Staubli VAL3: InitBelt.pgx

program InitBelt()
begin
  //砂带信息初始化
  nPYC=0
  nPY=0
  nPYtest=0
  popUpMsg("砂带初始化完成!")
  logMsg("砂带初始化完成!")

end
